INTERFACE I_AlarmActions

METHOD Acknowledge : I_AlarmActionBy
VAR_INPUT
END_VAR
END_METHOD

METHOD Deactivate : I_AlarmActionBy
VAR_INPUT
END_VAR
END_METHOD

METHOD Raise : I_AlarmActionBy
VAR_INPUT
END_VAR
END_METHOD

END_INTERFACE

(* stored: Version 1.1.0.1, ProductVersion 3.1.4024.13
   Itf I_AlarmActions: Id {6fe788ed-b8fe-037d-186b-e4a0a1d8baaf}
   Method Acknowledge: Id {a835e518-0661-094a-227c-8a35d7d52de8}
   Method Deactivate: Id {c42eb63c-f69e-057b-1915-2340ce3be9f0}
   Method Raise: Id {5760bf2f-a9dd-01b1-1d16-fcc4cdc7ac11} *)
